(* Logix 5000 project; controller Transcat_L33ER vendor 1 type 14 code 107 rev 32.11; software revision 32.02; part 3 of 4 *)
(* tags used below, declared in another part *)
   AllDevice1stScanDone : BOOL;   // When this bit is set - all devices have been scanned once and bits reset
   alwaysOFF : BOOL;
   AnyAutoDeviceInterlock : BOOL;   // Any device in Auto interlocked
   AnyAutoRun : BOOL;   // Bit that in on if ANY device is placed into Auto run (to signal pre-start beed)
   AnyAutoRunFlag : BOOL;   // A flag that indicates if any device is in Auto Run (used with pre-start beep logic)
   AnyDeviceInterlock : BOOL;   // Any device is interlocked
   AnyManRunFlag : BOOL;   // A flag that indicates if any device is in Manual Run (used with pre-start beep logic)
   AnyManualRun : BOOL;   // Bit that in on if ANY device is placed into manual run (to signal pre-start beed)
   Auto_Run_All_Interlock : BOOL;   // Bit to interlock all devices running in Auto
   BeaconBlueLight : ALIAS FOR TC_Remote_IO:3:O.3;   // Blue Beacon Light
   BeaconGreenLight : ALIAS FOR TC_Remote_IO:3:O.2;   // Green Beacon Light
   BeaconRedLight : ALIAS FOR TC_Remote_IO:3:O.0;   // Red Beacon Light
   BeaconYellowLight : ALIAS FOR TC_Remote_IO:3:O.1;   // Yellow Beacon Light
   Beep : BOOL;   // Bit to Activte Beacon Alarm
   BeepNew : ALIAS FOR TC_Remote_IO:3:O.4;
   Device : Device[20];
   DiscreteTemp : BOOL;   // A temporay boolean to hold positions during PLC transer
   dNum : DINT;   // The index of the current device being processed
   DoseCounter : COUNTER;   // Counts the # of doses since last reset
   DoseCounterReset_HMI : BOOL;   // HMI bit to reset the dose counter
   DoseStart : BOOL;   // Bit to start dosing sequence
   DoseStartOneShot : BOOL;   // One shot to start dosing
   DoseStop : BOOL;   // Bit to stop dosing
   DoseStopOneShot : BOOL;   // one shot to stop dosing
   DoseTarget : REAL;   // Target dose amount
   FT103 : BronkhorstFlowMeter;
   FT103B : BronkhorstFlowMeter;
   FT104 : BronkhorstFlowMeter;
   FT104B : BronkhorstFlowMeter;
   FT105 : BronkhorstFlowMeter;
   FT105B : BronkhorstFlowMeter;
   GF101 : Thayer_WB_Feeder;   // Thayer 1 Tags
   GF201 : Thayer_WB_Feeder;   // Thayer 2 Tags
   GF201_Totalizer1 : ALIAS FOR Thayer2Data[9];   // Thayer 2 (GF201) Totalizer 1 in lbs
   GF201_Write_Total1Reset : ALIAS FOR Thayer2_BS:O.Data[2].1;   // Thayer 2 (GF1201) Totalizer 1 reset
   GF301 : Acrison_Feeder;   // GF103 - Small Feeder 1
   GreenFlashingOff : TIMER;
   GreenFlashingOn : TIMER;
   HMI_AllReset : BOOL;   // Bit to reset Auto/Man, AutoRun, RecipeRun, TimedRunEnable to 0 from HMI
   HMI_ProcessReset : BOOL;   // Bit to clear the process hold/inteerlock when all other device interlocks are cleared
   InitCount : INT;   // Counter to cycle through each device on start-up and reset AutoMan, AutoRun, ManualRun bits
   MSG_FROM_SLC500 : INT[10];
   MX101 : Howes_Mixer;
   MX201 : Howes_Mixer;
   PT103_PV_RAW : ALIAS FOR TC_Remote_IO:1:I.Ch0Data;   // Raw (unscaled) pressure reading from PT103 - PSI * 100 (range 0 - 108 PSI)
   PT104_PV_RAW : ALIAS FOR TC_Remote_IO:1:I.Ch1Data;   // Raw (unscaled) pressure reading from PT104 - PSI * 100 (range 0 - 108 PSI)
   PT105_PV_RAW : ALIAS FOR TC_Remote_IO:1:I.Ch2Data;   // Raw (unscaled) pressure reading from PT105 - PSI * 100 (range 0 - 108 PSI)
   StartBeepTimer : TIMER;   // Timer to sound the beep alarm before starting a device
   Thayer2ResetTotal1_HMI : BOOL;   // Bit to reset Thayer2 - totalizer 1 from HMI
   UpperHowesSpeed : INT;
   VF101 : Acrison_Feeder;   // Medium Feeder Tags
   VF201 : Acrison_Feeder;   // Small Feeder 2 Tags
   YellowFlashOff : TIMER;
   YellowFlashOn : TIMER;
(* MainProgram, continued *)

ROUTINE DeviceManager   (* ladder *)
// Loop through all devices each scan
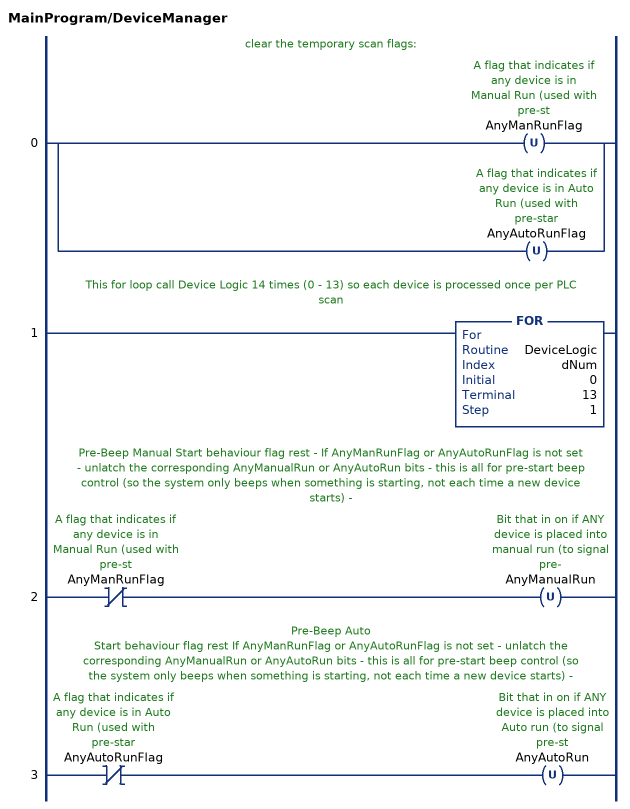
   // clear the temporary scan flags:
   0: [OTU(AnyManRunFlag) ,OTU(AnyAutoRunFlag) ];
   // This for loop call Device Logic 14 times (0 - 13) so each device is processed once per PLC scan
   1: FOR(DeviceLogic,dNum,0,13,1);
   // Pre-Beep Manual Start behaviour flag rest - If AnyManRunFlag or AnyAutoRunFlag is not set - unlatch the corresponding AnyManualRun or AnyAutoRun bits - this is all for pre-start beep control (so the system only beeps when something is starting, not each time a new device starts) -
   2: XIO(AnyManRunFlag)OTU(AnyManualRun);
   // Pre-Beep Auto
   //  Start behaviour flag rest If AnyManRunFlag or AnyAutoRunFlag is not set - unlatch the corresponding AnyManualRun or AnyAutoRun bits - this is all for pre-start beep control (so the system only beeps when something is starting, not each time a new device starts) -
   3: XIO(AnyAutoRunFlag)OTU(AnyAutoRun);
END_ROUTINE

ROUTINE GF201Dose   (* ladder *)
// Logic to Dose a specific amount from GF201 - Thayer 2
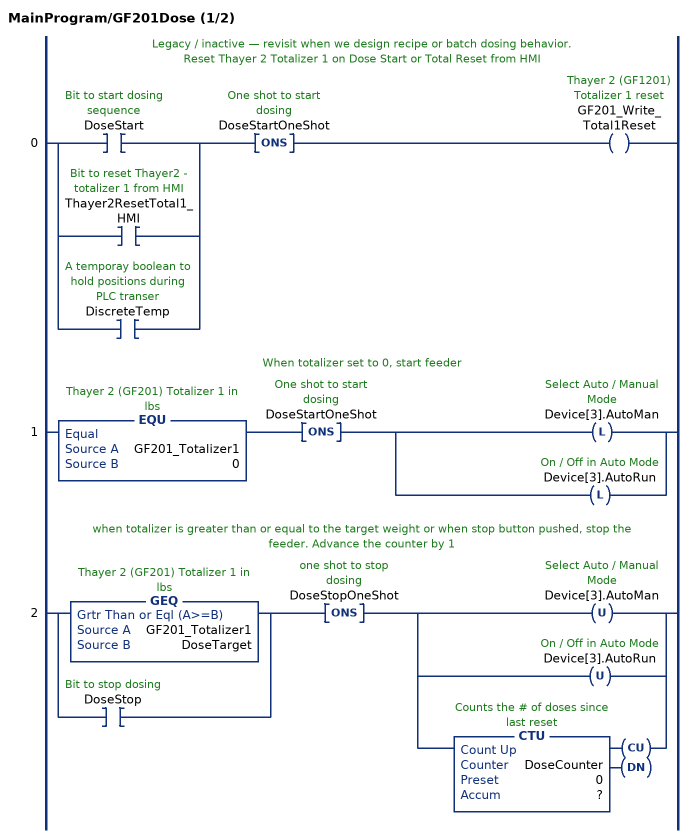
   // Legacy / inactive — revisit when we design recipe or batch dosing behavior.
   // Reset Thayer 2 Totalizer 1 on Dose Start or Total Reset from HMI
   0: [XIC(DoseStart) ,[XIC(Thayer2ResetTotal1_HMI) ,XIC(DiscreteTemp) ] ]ONS(DoseStartOneShot)OTE(GF201_Write_Total1Reset);
   // When totalizer set to 0, start feeder
   1: EQU(GF201_Totalizer1,0)ONS(DoseStartOneShot)[OTL(Device[3].AutoMan) ,OTL(Device[3].AutoRun) ];
   // when totalizer is greater than or equal to the target weight or when stop button pushed, stop the feeder. Advance the counter by 1
   2: [GEQ(GF201_Totalizer1,DoseTarget) ,XIC(DoseStop) ]ONS(DoseStopOneShot)[OTU(Device[3].AutoMan) ,[OTU(Device[3].AutoRun) ,CTU(DoseCounter,?,?) ] ];
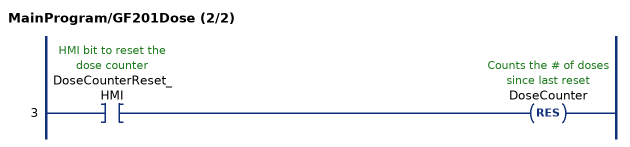
   3: XIC(DoseCounterReset_HMI)RES(DoseCounter);
END_ROUTINE

ROUTINE Initialize   (* ladder *)
// Reset controls and any other initialization required
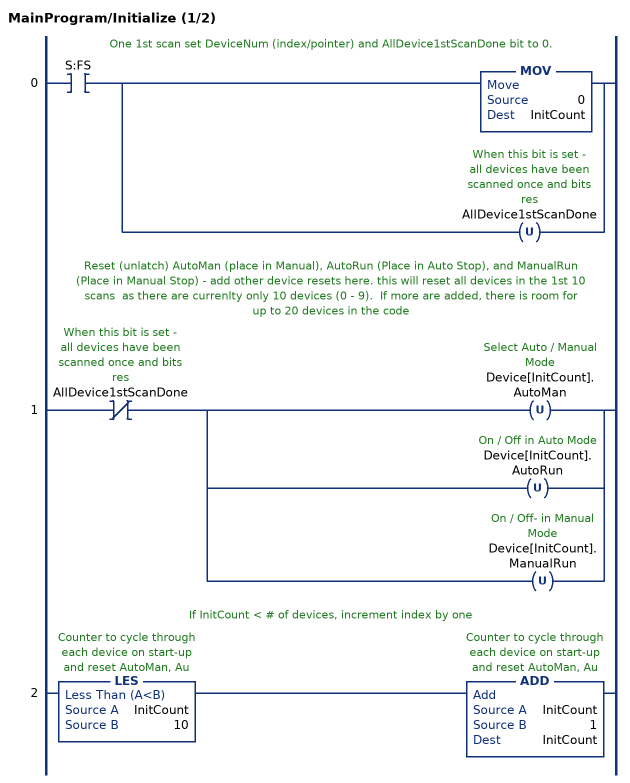
   // One 1st scan set DeviceNum (index/pointer) and AllDevice1stScanDone bit to 0.
   0: XIC(S:FS)[MOV(0,InitCount) ,OTU(AllDevice1stScanDone) ];
   // Reset (unlatch) AutoMan (place in Manual), AutoRun (Place in Auto Stop), and ManualRun (Place in Manual Stop) - add other device resets here. this will reset all devices in the 1st 10 scans  as there are currenlty only 10 devices (0 - 9).  If more are added, there is room for up to 20 devices in the code
   1: XIO(AllDevice1stScanDone)[OTU(Device[InitCount].AutoMan) ,[OTU(Device[InitCount].AutoRun) ,OTU(Device[InitCount].ManualRun) ] ];
   // If InitCount < # of devices, increment index by one
   2: LES(InitCount,10)ADD(InitCount,1,InitCount);
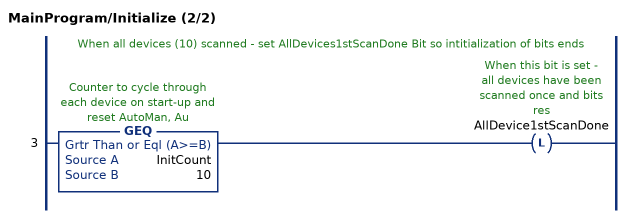
   // When all devices (10) scanned - set AllDevices1stScanDone Bit so intitialization of bits ends
   3: GEQ(InitCount,10)OTL(AllDevice1stScanDone);
END_ROUTINE

ROUTINE InterlockLogic   (* ladder *)
// All interlock logic is handled here
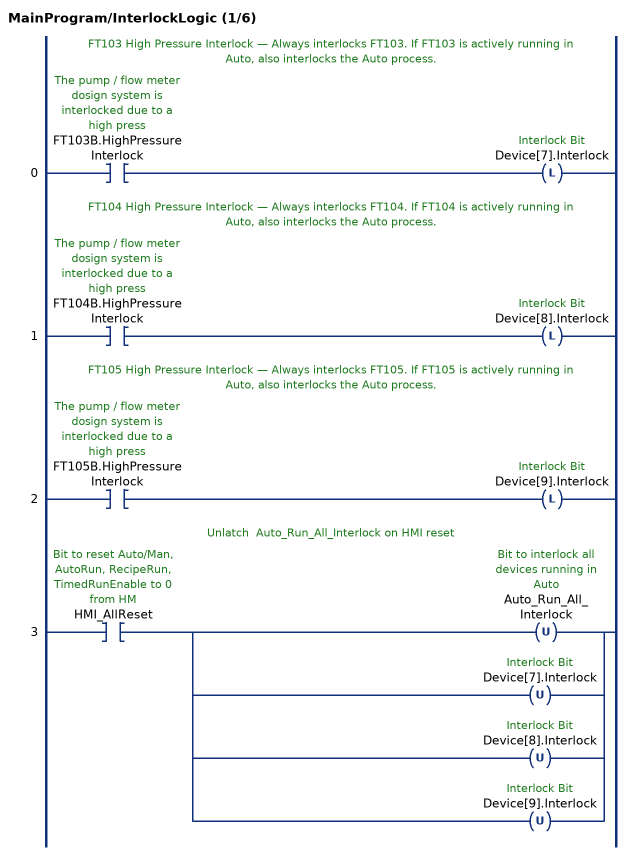
   // FT103 High Pressure Interlock — Always interlocks FT103. If FT103 is actively running in Auto, also interlocks the Auto process.
   0: XIC(FT103B.HighPressureInterlock)OTL(Device[7].Interlock);
   // FT104 High Pressure Interlock — Always interlocks FT104. If FT104 is actively running in Auto, also interlocks the Auto process.
   1: XIC(FT104B.HighPressureInterlock)OTL(Device[8].Interlock);
   // FT105 High Pressure Interlock — Always interlocks FT105. If FT105 is actively running in Auto, also interlocks the Auto process.
   2: XIC(FT105B.HighPressureInterlock)OTL(Device[9].Interlock);
   // Unlatch  Auto_Run_All_Interlock on HMI reset
   3: XIC(HMI_AllReset)[OTU(Auto_Run_All_Interlock) ,[OTU(Device[7].Interlock) ,[OTU(Device[8].Interlock) ,OTU(Device[9].Interlock) ] ] ];
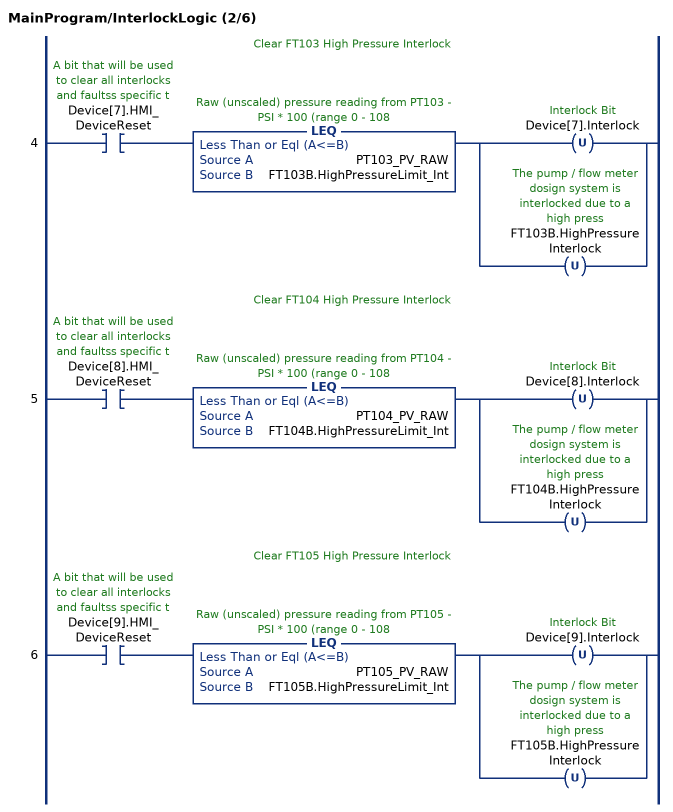
   // Clear FT103 High Pressure Interlock
   4: XIC(Device[7].HMI_DeviceReset)LEQ(PT103_PV_RAW,FT103B.HighPressureLimit_Int)[OTU(Device[7].Interlock) ,OTU(FT103B.HighPressureInterlock) ];
   // Clear FT104 High Pressure Interlock
   5: XIC(Device[8].HMI_DeviceReset)LEQ(PT104_PV_RAW,FT104B.HighPressureLimit_Int)[OTU(Device[8].Interlock) ,OTU(FT104B.HighPressureInterlock) ];
   // Clear FT105 High Pressure Interlock
   6: XIC(Device[9].HMI_DeviceReset)LEQ(PT105_PV_RAW,FT105B.HighPressureLimit_Int)[OTU(Device[9].Interlock) ,OTU(FT105B.HighPressureInterlock) ];
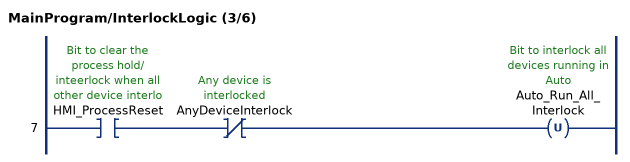
   7: XIC(HMI_ProcessReset)XIO(AnyDeviceInterlock)OTU(Auto_Run_All_Interlock);
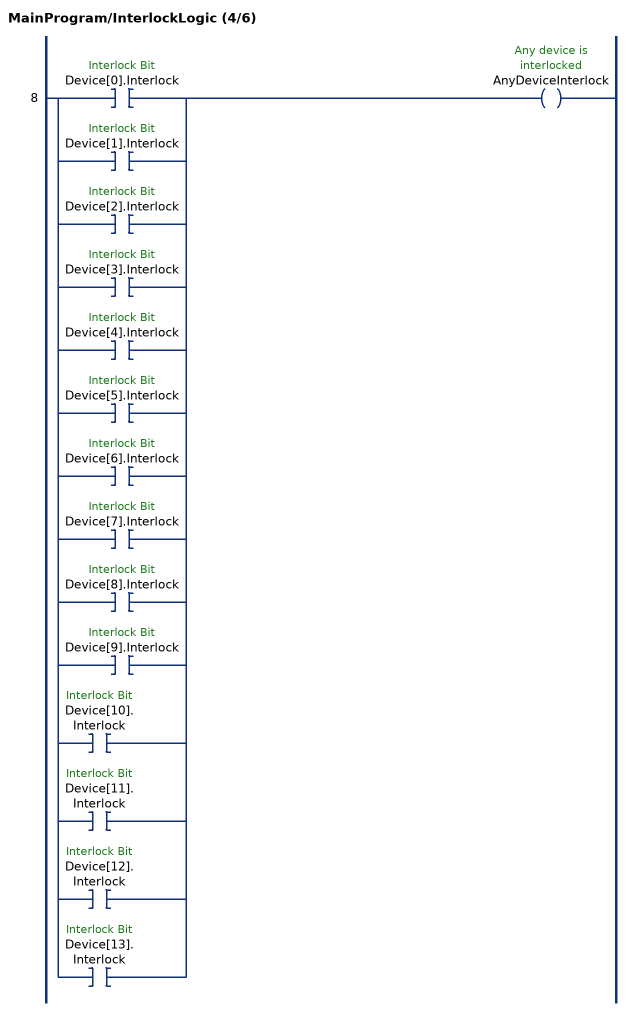
   8: [XIC(Device[0].Interlock) ,XIC(Device[1].Interlock) ,XIC(Device[2].Interlock) ,XIC(Device[3].Interlock) ,XIC(Device[4].Interlock) ,XIC(Device[5].Interlock) ,XIC(Device[6].Interlock) ,XIC(Device[7].Interlock) ,XIC(Device[8].Interlock) ,XIC(Device[9].Interlock) ,XIC(Device[10].Interlock) ,XIC(Device[11].Interlock) ,XIC(Device[12].Interlock) ,XIC(Device[13].Interlock) ]OTE(AnyDeviceInterlock);
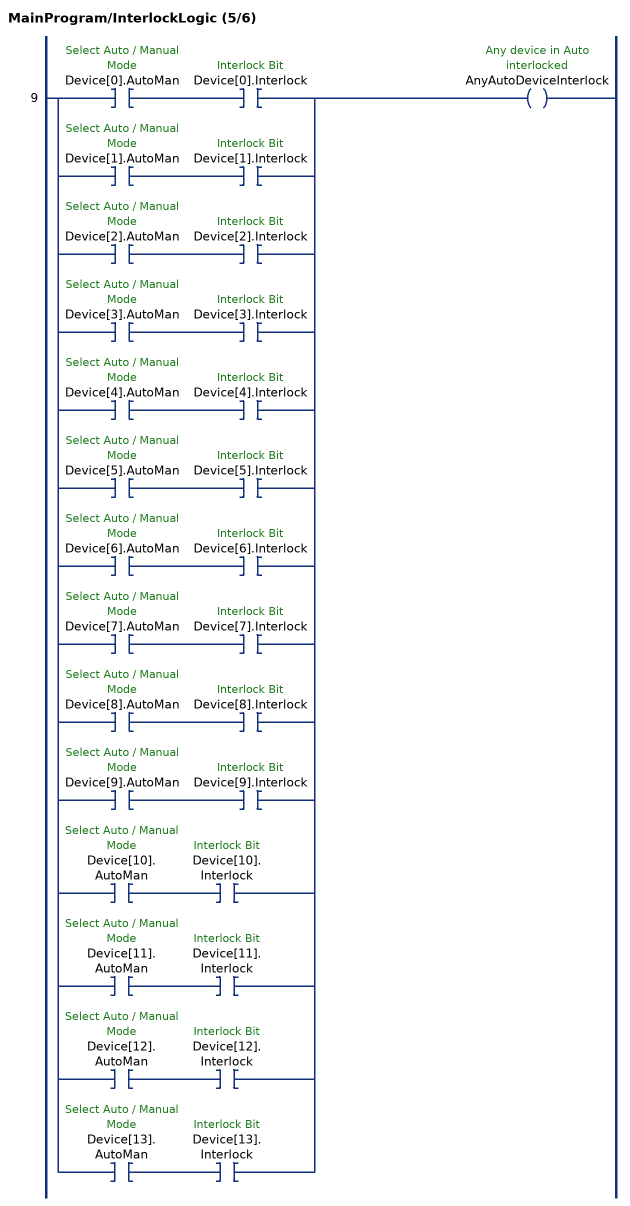
   9: [XIC(Device[0].AutoMan) XIC(Device[0].Interlock) ,XIC(Device[1].AutoMan) XIC(Device[1].Interlock) ,XIC(Device[2].AutoMan) XIC(Device[2].Interlock) ,XIC(Device[3].AutoMan) XIC(Device[3].Interlock) ,XIC(Device[4].AutoMan) XIC(Device[4].Interlock) ,XIC(Device[5].AutoMan) XIC(Device[5].Interlock) ,XIC(Device[6].AutoMan) XIC(Device[6].Interlock) ,XIC(Device[7].AutoMan) XIC(Device[7].Interlock) ,XIC(Device[8].AutoMan) XIC(Device[8].Interlock) ,XIC(Device[9].AutoMan) XIC(Device[9].Interlock) ,XIC(Device[10].AutoMan) XIC(Device[10].Interlock) ,XIC(Device[11].AutoMan) XIC(Device[11].Interlock) ,XIC(Device[12].AutoMan) XIC(Device[12].Interlock) ,XIC(Device[13].AutoMan) XIC(Device[13].Interlock) ]OTE(AnyAutoDeviceInterlock);
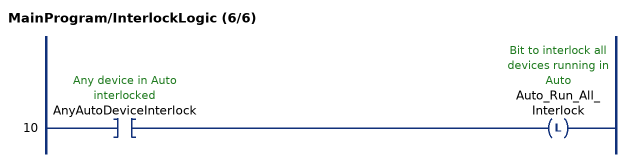
   10: XIC(AnyAutoDeviceInterlock)OTL(Auto_Run_All_Interlock);
END_ROUTINE

ROUTINE Light_Beacon   (* ladder *)
// Indicator Light Beacon
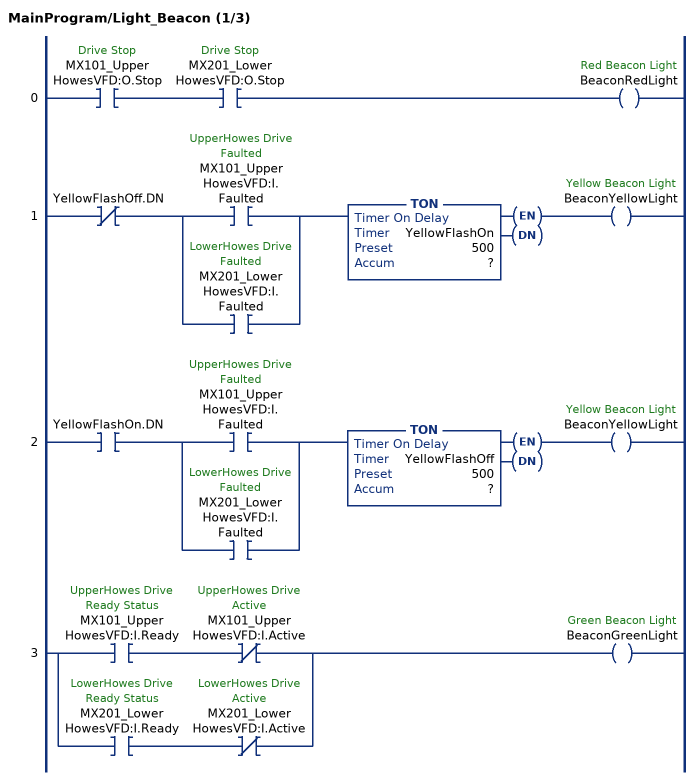
   0: XIC(MX101_UpperHowesVFD:O.Stop)XIC(MX201_LowerHowesVFD:O.Stop)OTE(BeaconRedLight);
   1: XIO(YellowFlashOff.DN)[XIC(MX101_UpperHowesVFD:I.Faulted) ,XIC(MX201_LowerHowesVFD:I.Faulted) ]TON(YellowFlashOn,?,?)OTE(BeaconYellowLight);
   2: XIC(YellowFlashOn.DN)[XIC(MX101_UpperHowesVFD:I.Faulted) ,XIC(MX201_LowerHowesVFD:I.Faulted) ]TON(YellowFlashOff,?,?)OTE(BeaconYellowLight);
   3: [XIC(MX101_UpperHowesVFD:I.Ready) XIO(MX101_UpperHowesVFD:I.Active) ,XIC(MX201_LowerHowesVFD:I.Ready) XIO(MX201_LowerHowesVFD:I.Active) ]OTE(BeaconGreenLight);
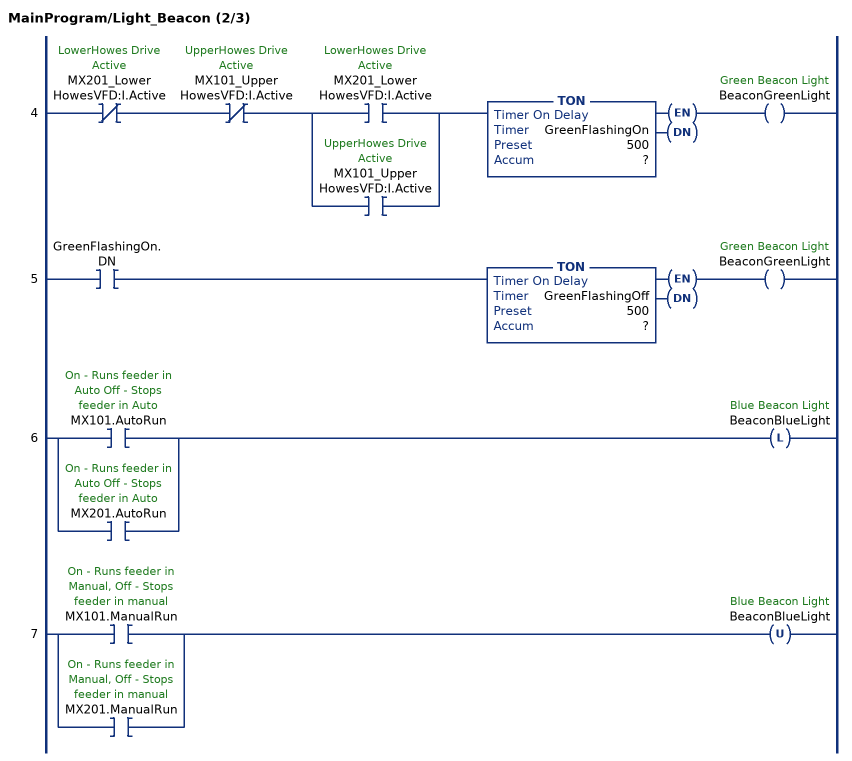
   4: XIO(MX201_LowerHowesVFD:I.Active)XIO(MX101_UpperHowesVFD:I.Active)[XIC(MX201_LowerHowesVFD:I.Active) ,XIC(MX101_UpperHowesVFD:I.Active) ]TON(GreenFlashingOn,?,?)OTE(BeaconGreenLight);
   5: XIC(GreenFlashingOn.DN)TON(GreenFlashingOff,?,?)OTE(BeaconGreenLight);
   6: [XIC(MX101.AutoRun) ,XIC(MX201.AutoRun) ]OTL(BeaconBlueLight);
   7: [XIC(MX101.ManualRun) ,XIC(MX201.ManualRun) ]OTU(BeaconBlueLight);
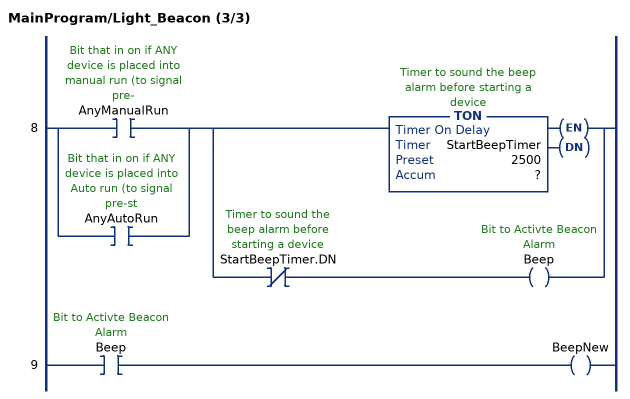
   8: [XIC(AnyManualRun) ,XIC(AnyAutoRun) ][TON(StartBeepTimer,?,?) ,XIO(StartBeepTimer.DN) OTE(Beep) ];
   9: XIC(Beep)OTE(BeepNew);
END_ROUTINE

ROUTINE MainRoutine   (* ladder *)
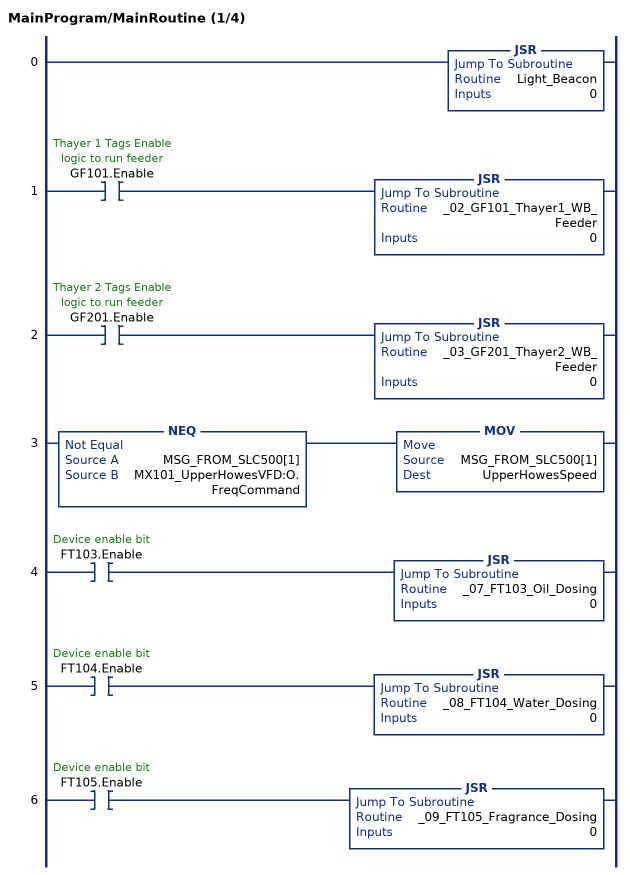
   0: JSR(Light_Beacon,0);
   1: XIC(GF101.Enable)JSR(_02_GF101_Thayer1_WB_Feeder,0);
   2: XIC(GF201.Enable)JSR(_03_GF201_Thayer2_WB_Feeder,0);
   3: NEQ(MSG_FROM_SLC500[1],MX101_UpperHowesVFD:O.FreqCommand)MOV(MSG_FROM_SLC500[1],UpperHowesSpeed);
   4: XIC(FT103.Enable)JSR(_07_FT103_Oil_Dosing,0);
   5: XIC(FT104.Enable)JSR(_08_FT104_Water_Dosing,0);
   6: XIC(FT105.Enable)JSR(_09_FT105_Fragrance_Dosing,0);
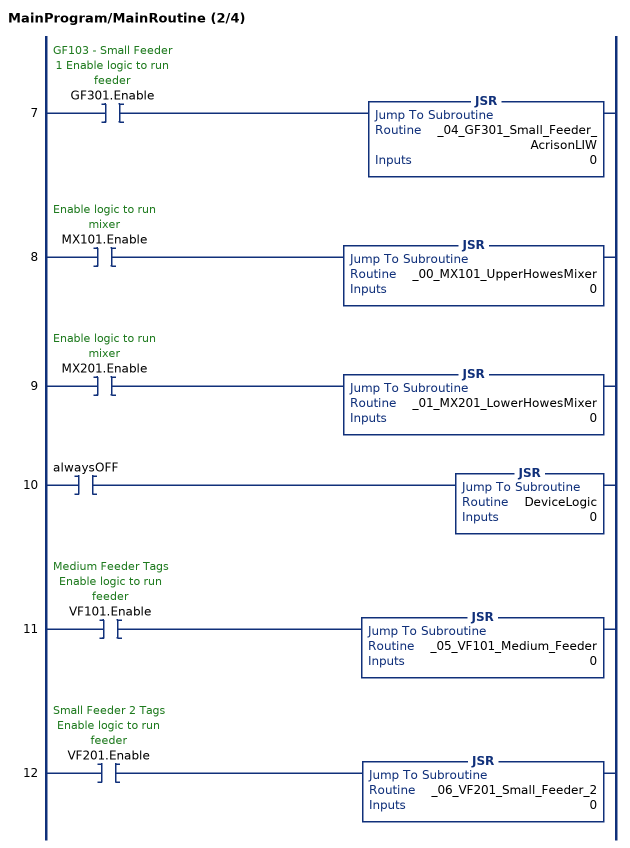
   7: XIC(GF301.Enable)JSR(_04_GF301_Small_Feeder_AcrisonLIW,0);
   8: XIC(MX101.Enable)JSR(_00_MX101_UpperHowesMixer,0);
   9: XIC(MX201.Enable)JSR(_01_MX201_LowerHowesMixer,0);
   10: XIC(alwaysOFF)JSR(DeviceLogic,0);
   11: XIC(VF101.Enable)JSR(_05_VF101_Medium_Feeder,0);
   12: XIC(VF201.Enable)JSR(_06_VF201_Small_Feeder_2,0);
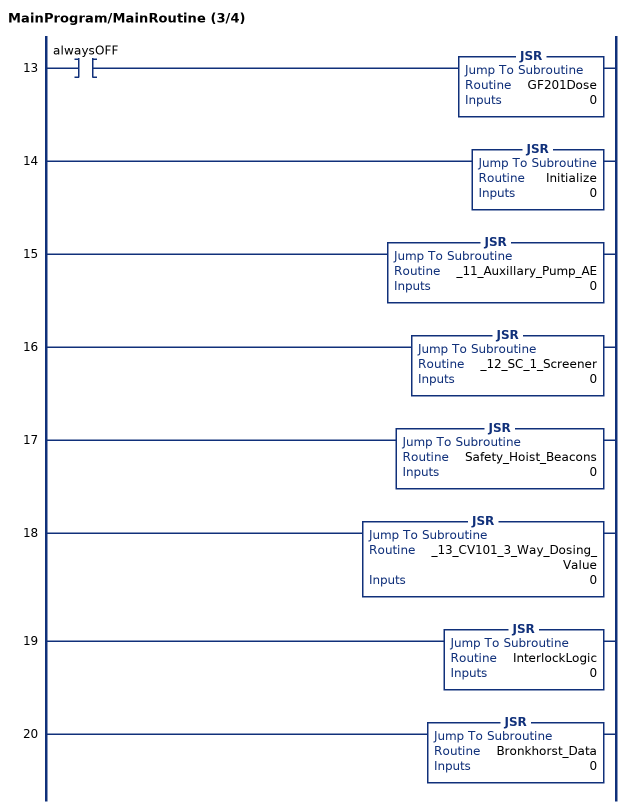
   13: XIC(alwaysOFF)JSR(GF201Dose,0);
   14: JSR(Initialize,0);
   15: JSR(_11_Auxillary_Pump_AE,0);
   16: JSR(_12_SC_1_Screener,0);
   17: JSR(Safety_Hoist_Beacons,0);
   18: JSR(_13_CV101_3_Way_Dosing_Value,0);
   19: JSR(InterlockLogic,0);
   20: JSR(Bronkhorst_Data,0);
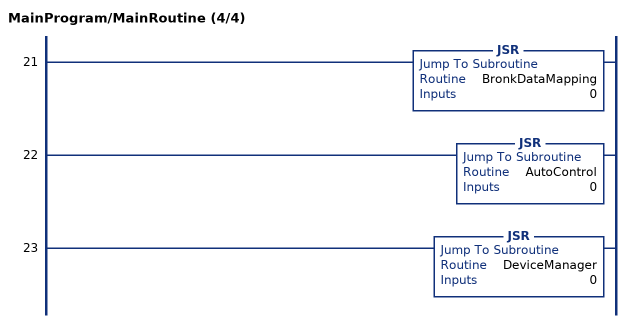
   21: JSR(BronkDataMapping,0);
   22: JSR(AutoControl,0);
   23: JSR(DeviceManager,0);
END_ROUTINE
